TYPE VEC3 :(* 3d position *)
STRUCT
	x, y, z : REAL;
END_STRUCT
END_TYPE

(* stored: Version 1.1.0.1, ProductVersion 3.1.0.25
   DUT VEC3: Id {6a672111-812a-471e-a05d-e3b015b100f8} *)
